KUKA KRL program: f_fraes1.src, f_fraes1.dat

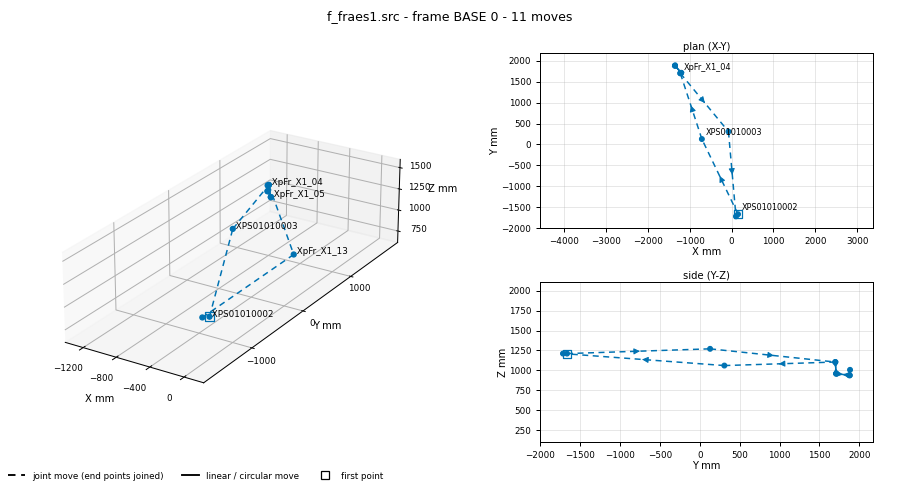
[picture p0: tool path of f_fraes1.src in frame BASE 0, 11 of 11 moves have a stored position in this frame; points joined in program order, loops and branches not executed]
--- f_fraes1.src ---
&ACCESS RVO3
&REL 6
&COMMENT INI Dress X1
&PARAM DISKPATH = KRC:\R1\Program
&PARAM TEMPLATE = C:\KRC\Roboter\Template\vorgabe
&PARAM EDITMASK = *
DEF f_fraes1( )
;FOLD INI
  ;FOLD BASISTECH INI
    GLOBAL INTERRUPT DECL 3 WHEN $STOPMESS==TRUE DO IR_STOPM ( )
    INTERRUPT ON 3
    BAS (#INITMOV,0 )
  ;ENDFOLD (BASISTECH INI)
;FOLD SPOTTECH INI
USERSPOT(#INIT)
;ENDFOLD (SPOTTECH INI)
;FOLD GRIPPERTECH INI
USER_GRP(0,DUMMY,DUMMY,GDEFAULT)
;ENDFOLD (GRIPPERTECH INI)
  ;FOLD USER INI
    ;Make your modifications here

  ;ENDFOLD (USER INI)
;ENDFOLD (INI)

; Caracterização dos meios de produção:
; Versão Atual:05/08/2015
; Name: P13.050-R2 CHANGES: Fresa X1
; (f2 6640 0018 985)



chk_w1_wechs_ok ( )    ; CHECK TOOL X1


;FOLD PTP PS01010002 CONT Vel=100 % PDAT18 Tool[1]:Gun X1 Base[0];%{PE}%R 8.2.20,%MKUKATPBASIS,%CMOVE,%VPTP,%P 1:PTP, 2:PS01010002, 3:C_DIS, 5:100, 7:PDAT18
$BWDSTART=FALSE
PDAT_ACT=PPDAT18
FDAT_ACT=FPS01010002
BAS(#PTP_PARAMS,100)
PTP XPS01010002 C_DIS
;ENDFOLD
;FOLD PTP PS01010003 CONT Vel=100 % PDAT19 Tool[1]:Gun X1 Base[0];%{PE}%R 8.2.20,%MKUKATPBASIS,%CMOVE,%VPTP,%P 1:PTP, 2:PS01010003, 3:C_DIS, 5:100, 7:PDAT19
$BWDSTART=FALSE
PDAT_ACT=PPDAT19
FDAT_ACT=FPS01010003
BAS(#PTP_PARAMS,100)
PTP XPS01010003 C_DIS
;ENDFOLD

;FOLD PTP pFr_X1_04 CONT Vel=100 % PDAT3 Tool[1]:Gun X1 Base[0];%{PE}%R 8.2.20,%MKUKATPBASIS,%CMOVE,%VPTP,%P 1:PTP, 2:pFr_X1_04, 3:C_DIS, 5:100, 7:PDAT3
$BWDSTART=FALSE
PDAT_ACT=PPDAT3
FDAT_ACT=FpFr_X1_04
BAS(#PTP_PARAMS,100)
PTP XpFr_X1_04 C_DIS
;ENDFOLD
;FOLD PTP pFr_X1_05 CONT Vel=100 % PDAT4 Tool[1]:Gun X1 Base[0];%{PE}%R 8.2.20,%MKUKATPBASIS,%CMOVE,%VPTP,%P 1:PTP, 2:pFr_X1_05, 3:C_DIS, 5:100, 7:PDAT4
$BWDSTART=FALSE
PDAT_ACT=PPDAT4
FDAT_ACT=FpFr_X1_05
BAS(#PTP_PARAMS,100)
PTP XpFr_X1_05 C_DIS
;ENDFOLD

;FOLD LIN pFr_X1_08 CONT Vel=1 m/s CPDAT1 Tool[1]:Gun X1 Base[0];%{PE}%R 8.2.20,%MKUKATPBASIS,%CMOVE,%VLIN,%P 1:LIN, 2:pFr_X1_08, 3:C_DIS C_DIS, 5:1, 7:CPDAT1
$BWDSTART=FALSE
LDAT_ACT=LCPDAT1
FDAT_ACT=FpFr_X1_08
BAS(#CP_PARAMS,1)
LIN XpFr_X1_08 C_DIS C_DIS
;ENDFOLD

;FOLD ; Ponto de fresagem;%{PE}%R 8.2.20,%MKUKATPBASIS,%CCOMMENT,%VNORMAL,%P 2:Ponto  de  fresagem
;ENDFOLD
;FOLD TIP.LIN_ Dress3, Spot Gun 4 , RETR open , Tool[1], Base[0], EXT.TCP=FALSE;%{PE}%MKUKATPUSER
FDAT_ACT=FDress3
BAS(#FRAMES)
LIN  XDress3
S_ACT.GUN=4
S_ACT.RETR=#opn
S_READY=FALSE
USERSPOT (#DRESS,S_ACT )
WAIT FOR  S_READY
;ENDFOLD

;FOLD LIN pFr_X1_10 CONT Vel=1 m/s CPDAT3 Tool[1]:Gun X1 Base[0];%{PE}%R 8.2.20,%MKUKATPBASIS,%CMOVE,%VLIN,%P 1:LIN, 2:pFr_X1_10, 3:C_DIS C_DIS, 5:1, 7:CPDAT3
$BWDSTART=FALSE
LDAT_ACT=LCPDAT3
FDAT_ACT=FpFr_X1_10
BAS(#CP_PARAMS,1)
LIN XpFr_X1_10 C_DIS C_DIS
;ENDFOLD

;FOLD PTP pFr_X1_007 PDAT17 SPOT Gun=4 RETR OPN PgNo1=254 ACTIVE=1 Tool[1]:Gun X1 Base[0];%{PE}%R 8.2.2,%MKUKATPSPOT,%CSPOT,%VPTP,%P 1:PTP, 2:pFr_X1_007, 3:, 5:100, 7:PDAT17, 10:4, 12:#FIRST, 14:#OPN, 16:254, 18:1, 20:0, 22:0, 24:1, 25:NORMAL
$BWDSTART=FALSE
PDAT_ACT=PPDAT17
FDAT_ACT=FpFr_X1_007
BAS(#PTP_PARAMS,PPDAT17.VEL)
S_ACT.GUN=4
S_ACT.PAIR=SDEFAULT.PAIR
S_ACT.RETR=#OPN
S_ACT.CLO_TM=1
S_ACT.PGNO1=254
S_ACT.PGNO2=SDEFAULT.PGNO2
S_ACT.PRESS1=SDEFAULT.PRESS1
S_ACT.PRESS2=SDEFAULT.PRESS2
S_READY=FALSE
PTP XpFr_X1_007
USERSPOT(#SPOT, S_ACT)
WAIT FOR S_READY
;ENDFOLD
;FOLD PTP pFr_X1_12 CONT Vel=100 % PDAT7 Tool[1]:Gun X1 Base[0];%{PE}%R 8.2.20,%MKUKATPBASIS,%CMOVE,%VPTP,%P 1:PTP, 2:pFr_X1_12, 3:C_DIS, 5:100, 7:PDAT7
$BWDSTART=FALSE
PDAT_ACT=PPDAT7
FDAT_ACT=FpFr_X1_12
BAS(#PTP_PARAMS,100)
PTP XpFr_X1_12 C_DIS
;ENDFOLD
;FOLD PTP pFr_X1_13 CONT Vel=100 % PDAT8 Tool[1]:Gun X1 Base[0];%{PE}%R 8.2.20,%MKUKATPBASIS,%CMOVE,%VPTP,%P 1:PTP, 2:pFr_X1_13, 3:C_DIS, 5:100, 7:PDAT8
$BWDSTART=FALSE
PDAT_ACT=PPDAT8
FDAT_ACT=FpFr_X1_13
BAS(#PTP_PARAMS,100)
PTP XpFr_X1_13 C_DIS
;ENDFOLD
;FOLD PTP pFr_X1_14 CONT Vel=100 % PDAT9 Tool[1]:Gun X1 Base[0];%{PE}%R 8.2.20,%MKUKATPBASIS,%CMOVE,%VPTP,%P 1:PTP, 2:pFr_X1_14, 3:C_DIS, 5:100, 7:PDAT9
$BWDSTART=FALSE
PDAT_ACT=PPDAT9
FDAT_ACT=FpFr_X1_14
BAS(#PTP_PARAMS,100)
PTP XpFr_X1_14 C_DIS
;ENDFOLD


END

--- f_fraes1.dat ---
&ACCESS RVO3
&REL 6
&COMMENT INI Dress X1
&PARAM DISKPATH = KRC:\R1\Program
&PARAM TEMPLATE = C:\KRC\Roboter\Template\vorgabe
&PARAM EDITMASK = *
DEFDAT  f_fraes1
;FOLD EXTERNAL DECLARATIONS;%{PE}%MKUKATPBASIS,%CEXT,%VCOMMON,%P
;FOLD GRIPPERTECH EXT
EXT  H50 (INT  :IN,INT  :IN,INT  :IN,GRP_TYP  :IN )
;ENDFOLD (GRIPPERTECH EXT)
;FOLD SPOTTECH EXT
EXT  USERSPOT (S_COMMAND  :IN,SPOT_TYPE  :IN )
;ENDFOLD (SPOTTECH EXT)
;FOLD BASISTECH EXT;%{PE}%MKUKATPBASIS,%CEXT,%VEXT,%P
EXT  BAS (BAS_COMMAND  :IN,REAL  :IN )
DECL INT SUCCESS
;ENDFOLD (BASISTECH EXT)
;FOLD USER EXT;%{E}%MKUKATPUSER,%CEXT,%VEXT,%P
;Make your modifications here

;ENDFOLD (USER EXT)
;ENDFOLD (EXTERNAL DECLARATIONS)
DECL BASIS_SUGG_T LAST_BASIS={POINT1[] "PS01010003              ",POINT2[] "PS01010003              ",CP_PARAMS[] "CPDAT0                  ",PTP_PARAMS[] "PDAT19                  ",CONT[] "C_DIS                   ",CP_VEL[] "2.0                     ",PTP_VEL[] "100                     ",SYNC_PARAMS[] "SYNCDAT                 ",SPL_NAME[] "S0                      "}
DECL PDAT PPDAT3={VEL 100.0,ACC 50.0,APO_DIST 50.0,APO_MODE #CDIS}
DECL E6POS XPFR_X1_04={X -1221.62195,Y 1698.92297,Z 1104.797,A 113.166603,B 33.5654984,C 7.35124302,S 6,T 26,E1 -1053.88599,E2 0.0,E3 0.0,E4 0.0,E5 0.0,E6 0.0}
DECL FDAT FpFr_X1_04={TOOL_NO 1,BASE_NO 0,IPO_FRAME #BASE,POINT2[] " ",TQ_STATE FALSE}
DECL PDAT PPDAT4={VEL 100.0,ACC 50.0,APO_DIST 50.0,APO_MODE #CDIS}
DECL E6POS XPFR_X1_05={X -1200.88696,Y 1709.09399,Z 959.197388,A 130.617401,B 5.28962803,C 1.01021099,S 6,T 18,E1 -1053.88501,E2 0.0,E3 0.0,E4 0.0,E5 0.0,E6 0.0}
DECL FDAT FpFr_X1_05={TOOL_NO 1,BASE_NO 0,IPO_FRAME #BASE,POINT2[] " ",TQ_STATE FALSE}
DECL LDAT LCPDAT1={VEL 2.0,ACC 100.0,APO_DIST 100.0,APO_FAC 50.0,AXIS_VEL 100.0,AXIS_ACC 100.0,ORI_TYP #VAR,CIRC_TYP #BASE,JERK_FAC 50.0,GEAR_JERK 50.0,EXAX_IGN 0}
DECL E6POS XPFR_X1_08={X -1346.94897,Y 1879.39697,Z 938.428284,A 130.617599,B 5.28952122,C 1.01018405,S 6,T 18,E1 -1053.88501,E2 0.0,E3 0.0,E4 0.0,E5 0.0,E6 0.0}
DECL FDAT FpFr_X1_08={TOOL_NO 1,BASE_NO 0,IPO_FRAME #BASE,POINT2[] " ",TQ_STATE FALSE}
DECL LDAT LCPDAT3={VEL 2.0,ACC 100.0,APO_DIST 100.0,APO_FAC 50.0,AXIS_VEL 100.0,AXIS_ACC 100.0,ORI_TYP #VAR,CIRC_TYP #BASE,JERK_FAC 50.0,GEAR_JERK 50.0,EXAX_IGN 0}
DECL E6POS XPFR_X1_10={X -1346.94604,Y 1879.39905,Z 938.425171,A 130.617401,B 5.28962803,C 1.01021099,S 6,T 18,E1 -1053.88501,E2 0.0,E3 0.0,E4 0.0,E5 0.0,E6 0.0}
DECL FDAT FpFr_X1_10={TOOL_NO 1,BASE_NO 0,IPO_FRAME #BASE,POINT2[] " ",TQ_STATE FALSE}
DECL PDAT PPDAT7={VEL 100.0,ACC 100.0,APO_DIST 100.0,APO_MODE #CDIS}
DECL E6POS XPFR_X1_12={X -1221.62195,Y 1698.92297,Z 1104.797,A 113.166603,B 33.5654984,C 7.35124302,S 6,T 26,E1 -1053.88599,E2 0.0,E3 0.0,E4 0.0,E5 0.0,E6 0.0}
DECL FDAT FpFr_X1_12={TOOL_NO 1,BASE_NO 0,IPO_FRAME #BASE,POINT2[] " ",TQ_STATE FALSE}
DECL PDAT PPDAT8={VEL 100.0,ACC 100.0,APO_DIST 100.0,APO_MODE #CDIS}
DECL E6POS XPFR_X1_13={X -73.0904465,Y 308.381897,Z 1060.63696,A 128.684692,B 83.8677902,C 120.861099,S 2,T 10,E1 -808.831421,E2 0.0,E3 0.0,E4 0.0,E5 0.0,E6 0.0}
DECL FDAT FpFr_X1_13={TOOL_NO 1,BASE_NO 0,IPO_FRAME #BASE,POINT2[] " ",TQ_STATE FALSE}
DECL PDAT PPDAT9={VEL 100.0,ACC 100.0,APO_DIST 100.0,APO_MODE #CDIS}
DECL E6POS XPFR_X1_14={X 106.391998,Y -1714.58203,Z 1210.95203,A -51.9155197,B 81.9439468,C 118.742798,S 2,T 10,E1 -808.812012,E2 0.0,E3 0.0,E4 0.0,E5 0.0,E6 0.0}
DECL FDAT FpFr_X1_14={TOOL_NO 1,BASE_NO 0,IPO_FRAME #BASE,POINT2[] " ",TQ_STATE FALSE}
DECL FDAT FDress3={TOOL_NO 1,BASE_NO 0,IPO_FRAME #BASE}
DECL E6POS XDress3={X -1348.98706,Y 1883.41602,Z 1007.04303,A 131.009003,B -1.36924195,C 0.477766097,S 6,T 18,E1 -1053.88,E2 0.0,E3 0.0,E4 0.0,E5 0.0,E6 0.0}
DECL SPOT_SUGG_T LAST_SPOT={GUN[] "1                       ",RETR_CMD[] "#OPN                    ",CHOISE[] "#FIRST                  ",CLO_TM[] "0                       ",PGNO1[] "1                       ",PRESS1[] "0                       ",PGNO2[] "1                       ",PRESS2[] "0                       ",SPOT_PARAMS[] "NORMAL                  "}
DECL PDAT PPDAT17={VEL 100.0,ACC 100.0,APO_DIST 100.0}
DECL E6POS XpFr_X1_007={X -1200.88904,Y 1709.09399,Z 959.199219,A 130.617493,B 5.28956985,C 1.01003301,S 6,T 18,E1 -1053.88501,E2 0.0,E3 0.0,E4 0.0,E5 0.0,E6 0.0}
DECL FDAT FpFr_X1_007={TOOL_NO 1,BASE_NO 0,IPO_FRAME #BASE,POINT2[] " ",TQ_STATE FALSE}
DECL E6POS XPS01010002={X 155.308807,Y -1663.75903,Z 1210.62,A -33.4589615,B 81.8930435,C 136.695602,S 2,T 10,E1 -808.810913,E2 0.0,E3 0.0,E4 0.0,E5 0.0,E6 0.0}
DECL FDAT FPS01010002={TOOL_NO 1,BASE_NO 0,IPO_FRAME #BASE,POINT2[] " ",TQ_STATE FALSE}
DECL PDAT PPDAT18={VEL 100.0,ACC 100.0,APO_DIST 100.0,APO_MODE #CDIS}
DECL E6POS XPS01010003={X -707.494995,Y 129.447601,Z 1270.31995,A 141.785904,B 72.6080933,C 102.7024,S 2,T 10,E1 -808.810608,E2 0.0,E3 0.0,E4 0.0,E5 0.0,E6 0.0}
DECL FDAT FPS01010003={TOOL_NO 1,BASE_NO 0,IPO_FRAME #BASE,POINT2[] " ",TQ_STATE FALSE}
DECL PDAT PPDAT19={VEL 100.0,ACC 100.0,APO_DIST 100.0,APO_MODE #CDIS}
ENDDAT
